// This function has been automatically generated from the project information.
{attribute 'signature_flag' := '1073741824'}
{attribute 'TcGenerated'}
{attribute 'no-analysis'}
FUNCTION F_GetVersion : ST_LibVersion
VAR_INPUT
	
END_VAR

F_GetVersion.iMajor := 1;
F_GetVersion.iMinor := 0;
F_GetVersion.iBuild := 0;
F_GetVersion.iRevision := 0;
F_GetVersion.sVersion := '1.0.0';
F_GetVersion.nFlags := 1;

END_FUNCTION

(* stored: Version 1.1.0.1
   POU F_GetVersion: Id {cb2afb79-9620-42b7-91af-f9c414b0bed4}, SpecialFunc None *)
